TYPE VirtualButtons :
STRUCT
	StartButton:BOOL;
	StopButton:BOOL;
	GroundButton:BOOL;
	AutomatButton:BOOL;

	StartLight : BOOL;
	StopLight : BOOL;
END_STRUCT
END_TYPE

(* stored: Version 1.1.0.1
   DUT VirtualButtons: Id {3425bad0-76df-4633-9294-0a58c68b91e0} *)
